(* Logix 5000 project; controller TBIL_All_AOIs_V0_3 vendor 1 type 14 code 176 rev 32.11; software revision 32.00; part 2 of 2 *)
(* tags used below, declared in another part *)
   TBEN_C_DATA : SINT[160];
   IOLDevice_PORT1 : BOOL;
   IOLDevice_PORT2 : BOOL;
   IOLDevice_PORT3 : BOOL;
   IOLDevice_PORT4 : BOOL;
   IOLDevice_PORT5 : BOOL;
   IOLDevice_PORT6 : BOOL;
   IOLDevice_PORT7 : BOOL;
   IOLDevice_PORT8 : BOOL;
   PORT5_Mode_IOL_or_DI : BOOL;   // 0: IO-LINK without validation 1: Port is set to DI (Power Cycle or Module Inhibit cycle require)
   PORT6_Mode_IOL_or_DI : BOOL;   // 0: IO-LINK without validation 1: Port is set to DI (Power Cycle or Module Inhibit cycle require)
   PORT7_Mode_IOL_or_DI : BOOL;   // 0: IO-LINK without validation 1: Port is set to DI (Power Cycle or Module Inhibit cycle require)
   PORT8_Mode_IOL_or_DI : BOOL;   // 0: IO-LINK without validation 1: Port is set to DI (Power Cycle or Module Inhibit cycle require)
   DisableOutput_DXP1 : BOOL;
   DisableOutput_DXP3 : BOOL;
   DisableOutput_DXP5 : BOOL;
   DisableOutput_DXP7 : BOOL;
   DeviceStatus : DINT;
   IOLReadActive : BOOL;
   IOLWriteActive : BOOL;
   IOL_READ_Request : BOOL;
   IOL_WRITE_Request : BOOL;
   Done : BOOL;
   Error : BOOL;
(* TBEN_Lx_8IOL_AOI, continued *)

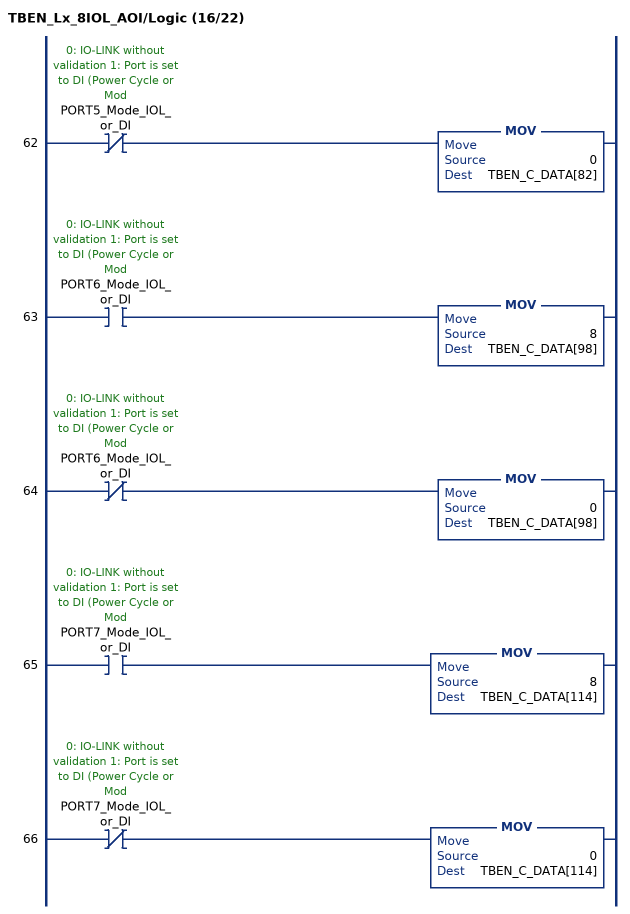
   62: XIO(PORT5_Mode_IOL_or_DI)MOV(0,TBEN_C_DATA[82]);
   63: XIC(PORT6_Mode_IOL_or_DI)MOV(8,TBEN_C_DATA[98]);
   64: XIO(PORT6_Mode_IOL_or_DI)MOV(0,TBEN_C_DATA[98]);
   65: XIC(PORT7_Mode_IOL_or_DI)MOV(8,TBEN_C_DATA[114]);
   66: XIO(PORT7_Mode_IOL_or_DI)MOV(0,TBEN_C_DATA[114]);
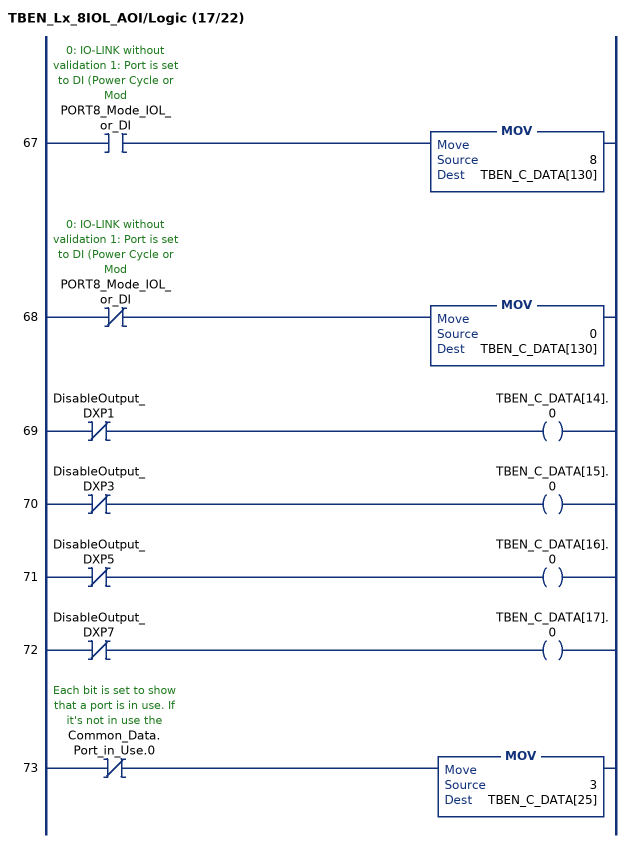
   67: XIC(PORT8_Mode_IOL_or_DI)MOV(8,TBEN_C_DATA[130]);
   68: XIO(PORT8_Mode_IOL_or_DI)MOV(0,TBEN_C_DATA[130]);
   69: XIO(DisableOutput_DXP1)OTE(TBEN_C_DATA[14].0);
   70: XIO(DisableOutput_DXP3)OTE(TBEN_C_DATA[15].0);
   71: XIO(DisableOutput_DXP5)OTE(TBEN_C_DATA[16].0);
   72: XIO(DisableOutput_DXP7)OTE(TBEN_C_DATA[17].0);
   73: XIO(Common_Data.Port_in_Use.0)MOV(3,TBEN_C_DATA[25]);
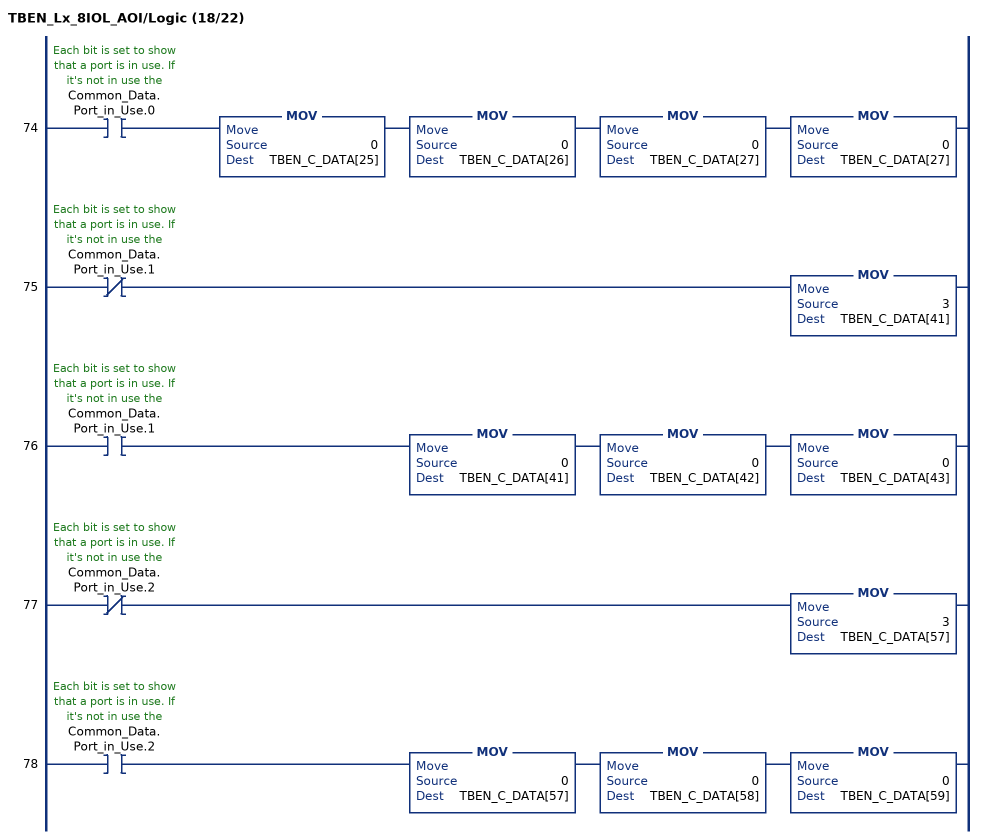
   74: XIC(Common_Data.Port_in_Use.0)MOV(0,TBEN_C_DATA[25])MOV(0,TBEN_C_DATA[26])MOV(0,TBEN_C_DATA[27])MOV(0,TBEN_C_DATA[27]);
   75: XIO(Common_Data.Port_in_Use.1)MOV(3,TBEN_C_DATA[41]);
   76: XIC(Common_Data.Port_in_Use.1)MOV(0,TBEN_C_DATA[41])MOV(0,TBEN_C_DATA[42])MOV(0,TBEN_C_DATA[43]);
   77: XIO(Common_Data.Port_in_Use.2)MOV(3,TBEN_C_DATA[57]);
   78: XIC(Common_Data.Port_in_Use.2)MOV(0,TBEN_C_DATA[57])MOV(0,TBEN_C_DATA[58])MOV(0,TBEN_C_DATA[59]);
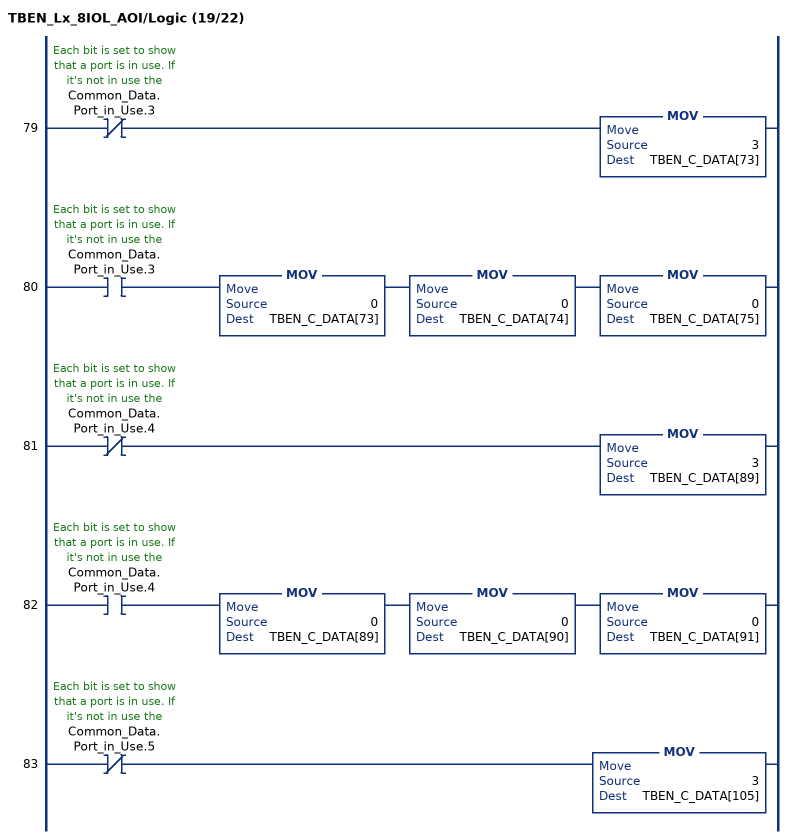
   79: XIO(Common_Data.Port_in_Use.3)MOV(3,TBEN_C_DATA[73]);
   80: XIC(Common_Data.Port_in_Use.3)MOV(0,TBEN_C_DATA[73])MOV(0,TBEN_C_DATA[74])MOV(0,TBEN_C_DATA[75]);
   81: XIO(Common_Data.Port_in_Use.4)MOV(3,TBEN_C_DATA[89]);
   82: XIC(Common_Data.Port_in_Use.4)MOV(0,TBEN_C_DATA[89])MOV(0,TBEN_C_DATA[90])MOV(0,TBEN_C_DATA[91]);
   83: XIO(Common_Data.Port_in_Use.5)MOV(3,TBEN_C_DATA[105]);
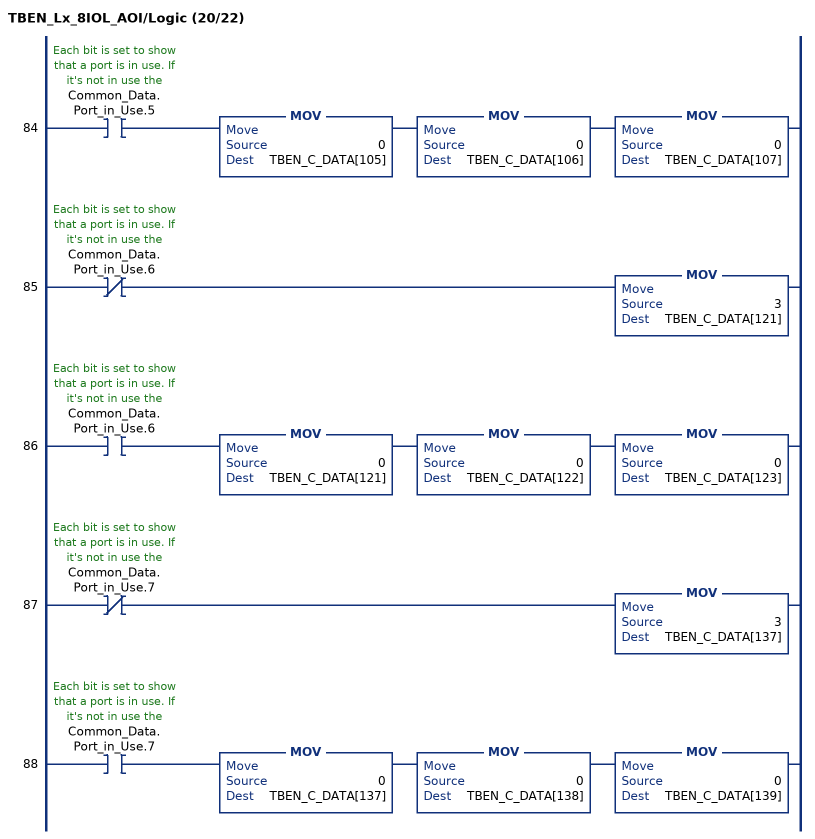
   84: XIC(Common_Data.Port_in_Use.5)MOV(0,TBEN_C_DATA[105])MOV(0,TBEN_C_DATA[106])MOV(0,TBEN_C_DATA[107]);
   85: XIO(Common_Data.Port_in_Use.6)MOV(3,TBEN_C_DATA[121]);
   86: XIC(Common_Data.Port_in_Use.6)MOV(0,TBEN_C_DATA[121])MOV(0,TBEN_C_DATA[122])MOV(0,TBEN_C_DATA[123]);
   87: XIO(Common_Data.Port_in_Use.7)MOV(3,TBEN_C_DATA[137]);
   88: XIC(Common_Data.Port_in_Use.7)MOV(0,TBEN_C_DATA[137])MOV(0,TBEN_C_DATA[138])MOV(0,TBEN_C_DATA[139]);
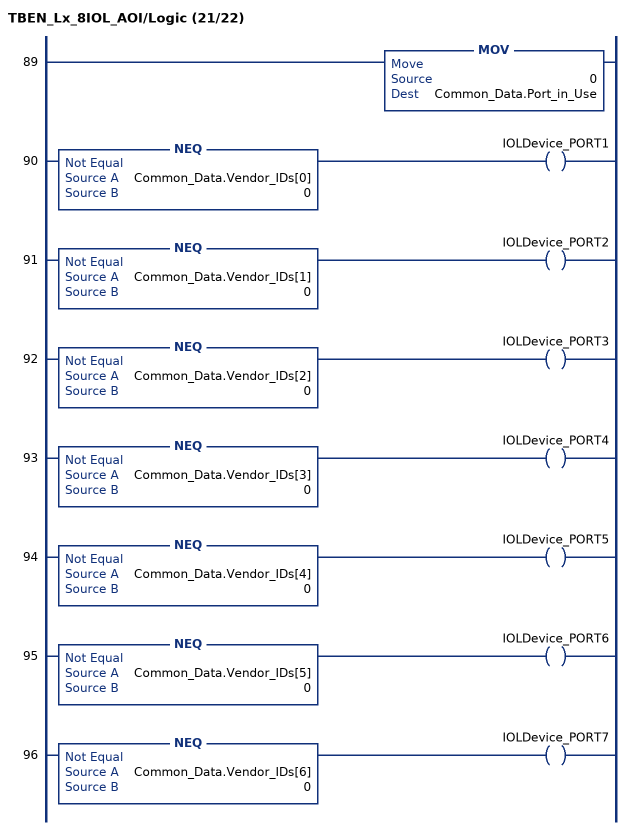
   89: MOV(0,Common_Data.Port_in_Use);
   90: NEQ(Common_Data.Vendor_IDs[0],0)OTE(IOLDevice_PORT1);
   91: NEQ(Common_Data.Vendor_IDs[1],0)OTE(IOLDevice_PORT2);
   92: NEQ(Common_Data.Vendor_IDs[2],0)OTE(IOLDevice_PORT3);
   93: NEQ(Common_Data.Vendor_IDs[3],0)OTE(IOLDevice_PORT4);
   94: NEQ(Common_Data.Vendor_IDs[4],0)OTE(IOLDevice_PORT5);
   95: NEQ(Common_Data.Vendor_IDs[5],0)OTE(IOLDevice_PORT6);
   96: NEQ(Common_Data.Vendor_IDs[6],0)OTE(IOLDevice_PORT7);
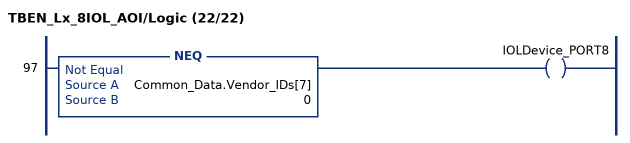
   97: NEQ(Common_Data.Vendor_IDs[7],0)OTE(IOLDevice_PORT8);
END_ROUTINE

ROUTINE Prescan   (* ladder *)
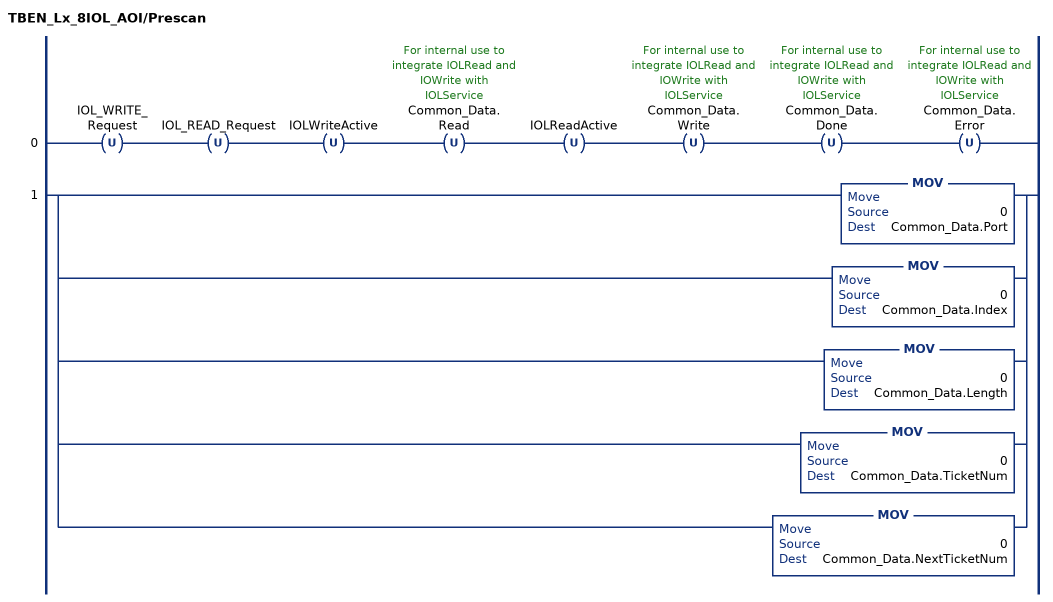
   0: OTU(IOL_WRITE_Request)OTU(IOL_READ_Request)OTU(IOLWriteActive)OTU(Common_Data.Read)OTU(IOLReadActive)OTU(Common_Data.Write)OTU(Common_Data.Done)OTU(Common_Data.Error);
   1: [MOV(0,Common_Data.Port) ,MOV(0,Common_Data.Index) ,MOV(0,Common_Data.Length) ,MOV(0,Common_Data.TicketNum) ,MOV(0,Common_Data.NextTicketNum) ];
END_ROUTINE
END_ADD_ON_INSTRUCTION

ADD_ON_INSTRUCTION Turck_TBIL_M1_16DXP_Full   (* revision 1.0 *)
VAR_INPUT
   Port : INT; {required}
END_VAR
VAR_IN_OUT
   Common_Data : Turck_IOLink_Common_Data; {required}
END_VAR
VAR_OUTPUT
   Input_1A : BOOL; {visible}
   Input_1B : BOOL; {visible}
   Input_2A : BOOL; {visible}
   Input_2B : BOOL; {visible}
   Input_3A : BOOL; {visible}
   Input_3B : BOOL; {visible}
   Input_4A : BOOL; {visible}
   Input_4B : BOOL; {visible}
   Input_5A : BOOL; {visible}
   Input_5B : BOOL; {visible}
   Input_6A : BOOL; {visible}
   Input_6B : BOOL; {visible}
   Input_7A : BOOL; {visible}
   Input_7B : BOOL; {visible}
   Input_8A : BOOL; {visible}
   Input_8B : BOOL; {visible}
END_VAR
VAR_INPUT
   Output_1A : BOOL; {visible}
   Output_1B : BOOL; {visible}
   Output_2A : BOOL; {visible}
   Output_2B : BOOL; {visible}
   Output_3A : BOOL; {visible}
   Output_3B : BOOL; {visible}
   Output_4A : BOOL; {visible}
   Output_4B : BOOL; {visible}
   Output_5A : BOOL; {visible}
   Output_5B : BOOL; {visible}
   Output_6A : BOOL; {visible}
   Output_6B : BOOL; {visible}
   Output_7A : BOOL; {visible}
   Output_7B : BOOL; {visible}
   Output_8A : BOOL; {visible}
   Output_8B : BOOL; {visible}
END_VAR
VAR_OUTPUT
   Wrong_or_Missing_Device : BOOL; {visible}
END_VAR
VAR
   Port_Less_One : INT; {access None}
   One : SINT; {access None}
   Port_Bit : SINT; {access None}
   Two : DINT; {access None}
END_VAR

ROUTINE Logic   (* ladder *)
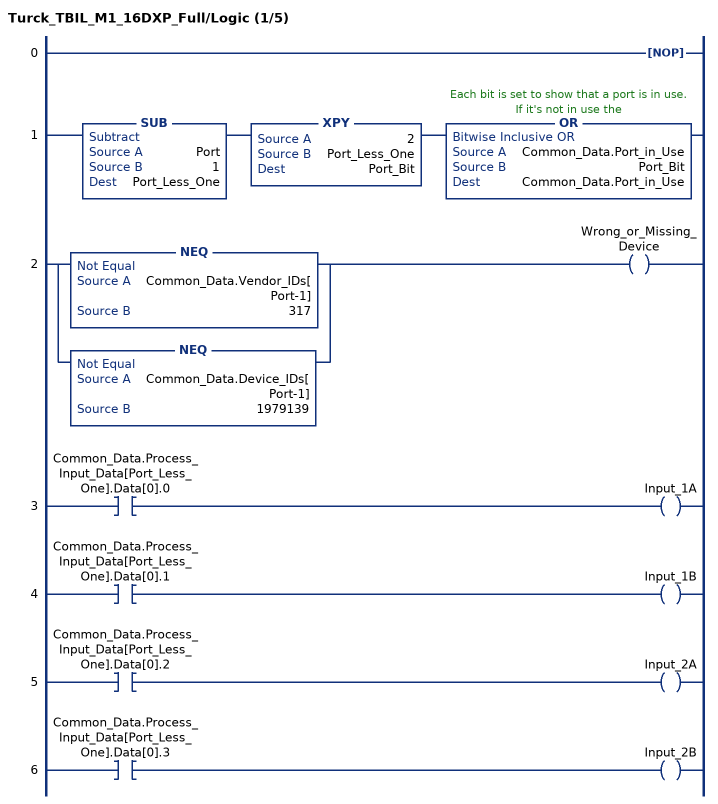
   0: NOP();
   1: SUB(Port,1,Port_Less_One)XPY(2,Port_Less_One,Port_Bit)OR(Common_Data.Port_in_Use,Port_Bit,Common_Data.Port_in_Use);
   2: [NEQ(Common_Data.Vendor_IDs[Port-1],317) ,NEQ(Common_Data.Device_IDs[Port-1],1979139) ]OTE(Wrong_or_Missing_Device);
   3: XIC(Common_Data.Process_Input_Data[Port_Less_One].Data[0].0)OTE(Input_1A);
   4: XIC(Common_Data.Process_Input_Data[Port_Less_One].Data[0].1)OTE(Input_1B);
   5: XIC(Common_Data.Process_Input_Data[Port_Less_One].Data[0].2)OTE(Input_2A);
   6: XIC(Common_Data.Process_Input_Data[Port_Less_One].Data[0].3)OTE(Input_2B);
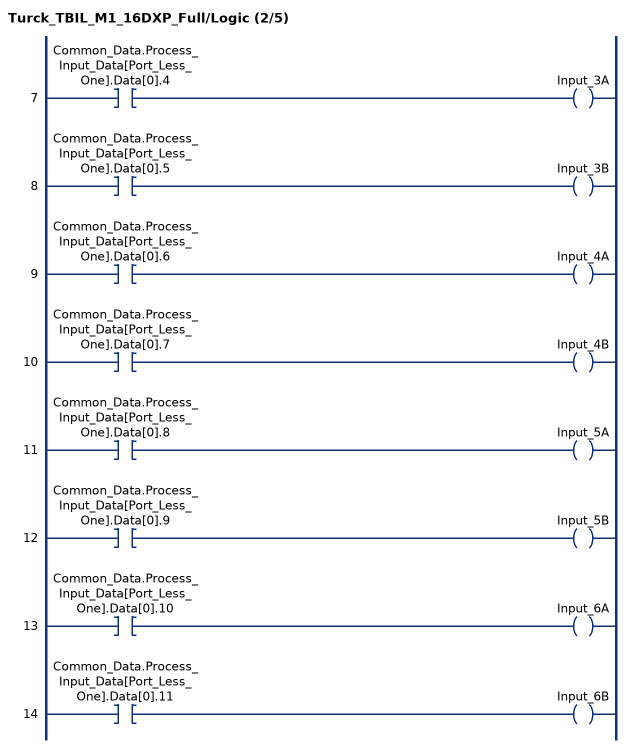
   7: XIC(Common_Data.Process_Input_Data[Port_Less_One].Data[0].4)OTE(Input_3A);
   8: XIC(Common_Data.Process_Input_Data[Port_Less_One].Data[0].5)OTE(Input_3B);
   9: XIC(Common_Data.Process_Input_Data[Port_Less_One].Data[0].6)OTE(Input_4A);
   10: XIC(Common_Data.Process_Input_Data[Port_Less_One].Data[0].7)OTE(Input_4B);
   11: XIC(Common_Data.Process_Input_Data[Port_Less_One].Data[0].8)OTE(Input_5A);
   12: XIC(Common_Data.Process_Input_Data[Port_Less_One].Data[0].9)OTE(Input_5B);
   13: XIC(Common_Data.Process_Input_Data[Port_Less_One].Data[0].10)OTE(Input_6A);
   14: XIC(Common_Data.Process_Input_Data[Port_Less_One].Data[0].11)OTE(Input_6B);
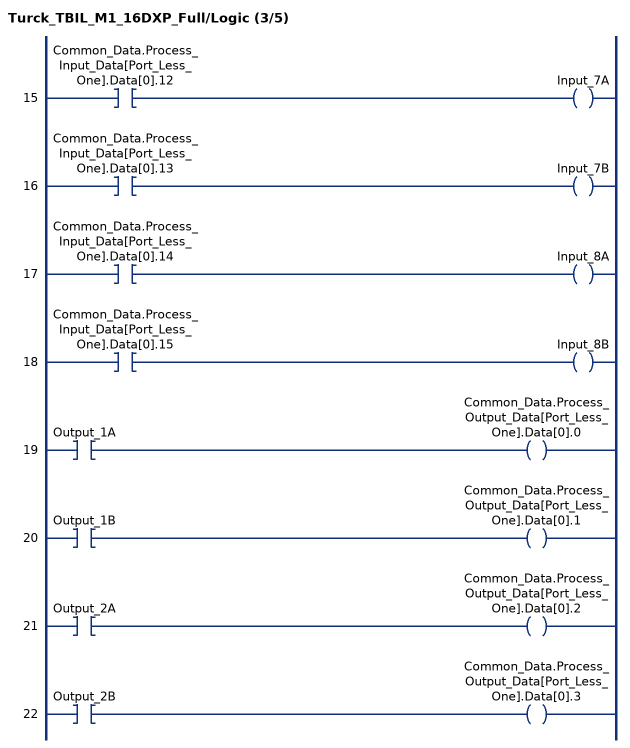
   15: XIC(Common_Data.Process_Input_Data[Port_Less_One].Data[0].12)OTE(Input_7A);
   16: XIC(Common_Data.Process_Input_Data[Port_Less_One].Data[0].13)OTE(Input_7B);
   17: XIC(Common_Data.Process_Input_Data[Port_Less_One].Data[0].14)OTE(Input_8A);
   18: XIC(Common_Data.Process_Input_Data[Port_Less_One].Data[0].15)OTE(Input_8B);
   19: XIC(Output_1A)OTE(Common_Data.Process_Output_Data[Port_Less_One].Data[0].0);
   20: XIC(Output_1B)OTE(Common_Data.Process_Output_Data[Port_Less_One].Data[0].1);
   21: XIC(Output_2A)OTE(Common_Data.Process_Output_Data[Port_Less_One].Data[0].2);
   22: XIC(Output_2B)OTE(Common_Data.Process_Output_Data[Port_Less_One].Data[0].3);
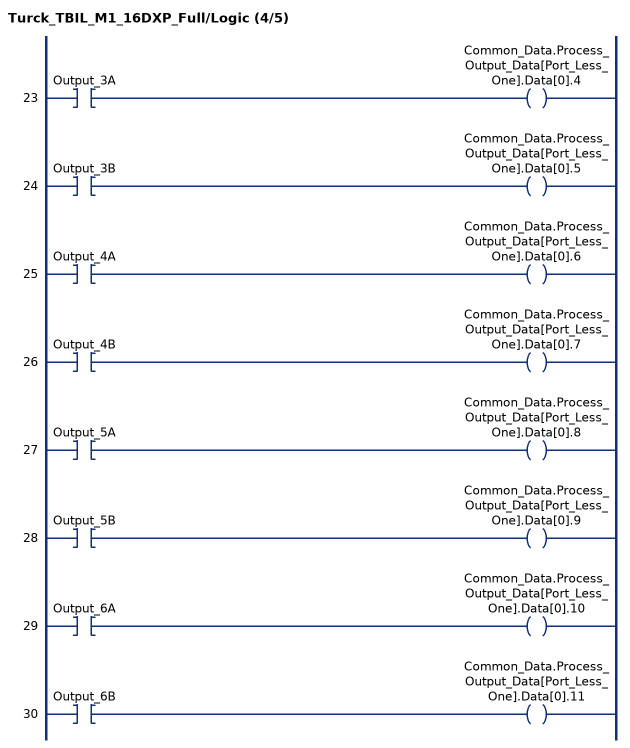
   23: XIC(Output_3A)OTE(Common_Data.Process_Output_Data[Port_Less_One].Data[0].4);
   24: XIC(Output_3B)OTE(Common_Data.Process_Output_Data[Port_Less_One].Data[0].5);
   25: XIC(Output_4A)OTE(Common_Data.Process_Output_Data[Port_Less_One].Data[0].6);
   26: XIC(Output_4B)OTE(Common_Data.Process_Output_Data[Port_Less_One].Data[0].7);
   27: XIC(Output_5A)OTE(Common_Data.Process_Output_Data[Port_Less_One].Data[0].8);
   28: XIC(Output_5B)OTE(Common_Data.Process_Output_Data[Port_Less_One].Data[0].9);
   29: XIC(Output_6A)OTE(Common_Data.Process_Output_Data[Port_Less_One].Data[0].10);
   30: XIC(Output_6B)OTE(Common_Data.Process_Output_Data[Port_Less_One].Data[0].11);
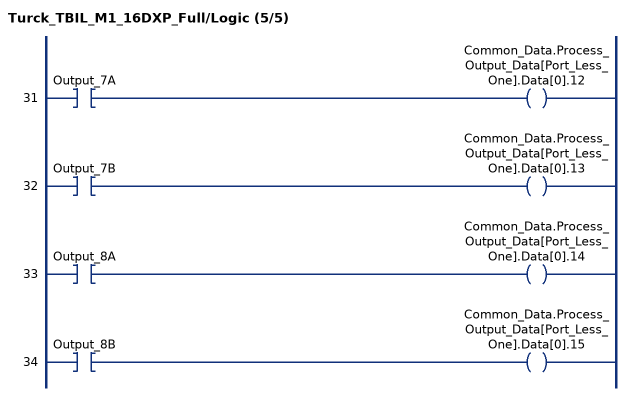
   31: XIC(Output_7A)OTE(Common_Data.Process_Output_Data[Port_Less_One].Data[0].12);
   32: XIC(Output_7B)OTE(Common_Data.Process_Output_Data[Port_Less_One].Data[0].13);
   33: XIC(Output_8A)OTE(Common_Data.Process_Output_Data[Port_Less_One].Data[0].14);
   34: XIC(Output_8B)OTE(Common_Data.Process_Output_Data[Port_Less_One].Data[0].15);
END_ROUTINE
END_ADD_ON_INSTRUCTION

VAR_GLOBAL   (* controller tags *)
   Common_Data : Turck_IOLink_Common_Data;
   IOL_READ_MSG : MESSAGE;
        MessageParameters(ServiceCode := 16#004b, LocalElement := Common_Data.SendData, DestinationTag := Common_Data.ReceiveData, ...)
   IOL_WRITE_MSG : MESSAGE;
        MessageParameters(ServiceCode := 16#004c, LocalElement := Common_Data.SendData, DestinationTag := Common_Data.ReceiveData, ...)
   TBEN_100_8IOL_AOI : TBEN_Lx_8IOL_AOI;
   TBIL_16DXP_AOI : Turck_TBIL_M1_16DXP_Full;
   TBIL_16DXP_Port_5 : IO_Link_Universal_Discrete_Hub;
END_VAR

PROGRAM MainProgram   (* main routine MainRoutine *)

ROUTINE MainRoutine   (* ladder *)
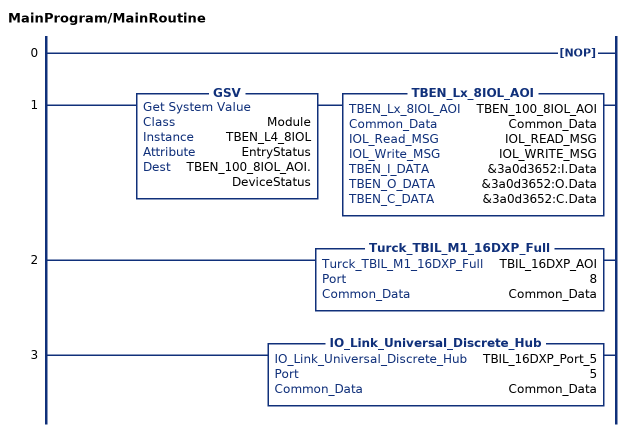
   0: NOP();
   1: GSV(Module,TBEN_L4_8IOL,EntryStatus,TBEN_100_8IOL_AOI.DeviceStatus)TBEN_Lx_8IOL_AOI(TBEN_100_8IOL_AOI,Common_Data,IOL_READ_MSG,IOL_WRITE_MSG,&3a0d3652:I.Data,&3a0d3652:O.Data,&3a0d3652:C.Data);
   2: Turck_TBIL_M1_16DXP_Full(TBIL_16DXP_AOI,8,Common_Data);
   3: IO_Link_Universal_Discrete_Hub(TBIL_16DXP_Port_5,5,Common_Data);
END_ROUTINE
END_PROGRAM

PROGRAM SafetyProgram   (* main routine MainRoutine, safety *)

ROUTINE MainRoutine   (* ladder *)
END_ROUTINE
END_PROGRAM
